// TwinCAT 3 PLC project PackMLtoTime
// ProgramVersion: 3.1.4023.0
// libraries:
//   Tc2_Standard, * (Beckhoff Automation GmbH)
//   Tc2_System, * (Beckhoff Automation GmbH)
//   Tc3_Module, * (Beckhoff Automation GmbH)
//   Tc3_PackML_V2, * (Beckhoff Automation GmbH)
//   Util, * (System)
// project tree:
//   / PlcTask.TcTTO
//   POUs/ daysInMonth.TcPOU, isLeapYear.TcPOU, MAIN.TcPOU, PakcML_TO_TIME.TcPOU
// real-time tasks:
//   TASK PlcTask: cycle T#10ms, priority 20, ADS port 350

CONFIGURATION PackMLtoTime
    RESOURCE PLC ON TwinCAT3
        TASK PlcTask(INTERVAL := T#10ms, PRIORITY := 20);
        PROGRAM MAIN WITH PlcTask : MAIN;
    END_RESOURCE
END_CONFIGURATION

// ---- POUs/MAIN.TcPOU
PROGRAM MAIN
VAR
	PackMLTime : ARRAY[0..6] OF DINT;
	bTest: BOOL;
	bTest2: BOOL;
	result: ULINT;
END_VAR

IF bTest THEN
	PackMLTime := ULINT_TO_PackMLTime(F_GetSystemTime());
END_IF

IF bTest2 THEN
	result := PakcML_TO_TIME(PackMLTime :=PackMLTime );
END_IF

END_PROGRAM

// ---- POUs/PakcML_TO_TIME.TcPOU
FUNCTION PakcML_TO_TIME : ULINT
VAR_INPUT
	PackMLTime	:	ARRAY[0..6] OF DINT;
END_VAR
VAR
	nYear: DINT;
	nMonth:DINT;
	nDay:DINT;
	nHour:DINT;
	nMinute: DINT;
	nSecond: DINT;
	nMiliSecond:DINT;
	uiMsCount: INT;
	nResult : ULINT;
END_VAR

nYear := PackMLTime[0];
nMonth := PackMLTime[1];
nDay := PackMLTime[2];
nHour := PackMLTime[3];
nMinute := PackMLTime[4];
nSecond := PackMLTime[5];
nMiliSecond := PackMLTime[6];

FOR uiMsCount := 1 TO 12 DO
	nResult := nResult + daysInMonth(nYear := DINT_TO_INT(nYear),nMonth:=uiMsCount);
END_FOR

nResult := (nResult *24 + nHour)*60+nMinute;
nResult := nResult * 60 + nSecond;
nResult := nResult*1000 + nMiliSecond;

END_FUNCTION

// ---- POUs/daysInMonth.TcPOU
FUNCTION daysInMonth : INT
VAR_INPUT
	nYear	: INT;
	nMonth	: INT;
END_VAR
VAR
END_VAR

CASE nMonth OF 
	1:
		daysInMonth := 31;
	2:
		daysInMonth := 28 + BOOL_TO_INT(isLeapYear(nYear:= nYear));
	3:
		daysInMonth := 31;
	4:
		daysInMonth := 30;
	5:
		daysInMonth := 31;
	6:
		daysInMonth := 30;
	7:
		daysInMonth := 31;
	8:
		daysInMonth := 31;
	9:
		daysInMonth := 30;
	10:
		daysInMonth := 31;
	11:
		daysInMonth := 30;
	12:
		daysInMonth := 31;
END_CASE

END_FUNCTION

// ---- POUs/isLeapYear.TcPOU
FUNCTION isLeapYear : Bool
VAR_INPUT
	nYear	: INT;
END_VAR
VAR
END_VAR

isLeapYear := (nYear / 4 = 0) AND (nYear / 100 <> 0) OR (nYear /400 = 0);

END_FUNCTION
